// TIA Portal V19 export
TYPE "LAF_typeDevDiagBasic"
TITLE = PN_DEV_DIAG
// This data type contains information for the HMI faceplate. / Autor: SICAR
// stored: Access Published
   STRUCT
      devNumber : UInt;   // Gerätenummer identisch mit Array-Index !!! / Device number, identical with array index !!!
      devName : String[24];   // Gerätename: ggf. WString, falls möglich; (SICAR: String24); 57 Zeichen sind in HW-Config eingebbar / Device name identified via "GET_NAME
      devStateDezCoded : USInt;   // Geräte-Status: dezimal codiert, zur einfachen Verwendung auf dem HMI / Device state decimal coded, for HMI animation
      devStateBitCoded : Word;   // Geräte-Status: Bit codiert, zur einfachen Verwendung auf dem HMI / Device state bit coded, for HMI animation
      first8CharOfMlfb : String[8];   // MLFB: ersten 8 Zeichen / First 8 characters of MLFB
   END_STRUCT;
END_TYPE
